
FUNCTION CB_dword_to_int : INT

TITLE = ' Convert a double word into an Integer '
VERSION : '1.0'
AUTHOR  : CB
NAME    : dworToIn
FAMILY  : TNI

VAR_INPUT
    IN : DWORD;
END_VAR

VAR_TEMP

END_VAR

BEGIN

CB_dword_to_int := DWORD_TO_INT(IN);

END_FUNCTION
